{attribute 'GeneratedUsingTerminal: EL2044-0000-0016'}
{attribute addProperty BoxType "EL2044-0000-0016"}
{attribute addProperty Id "Channel_1AT %Q*Channel_D623F56C1Channel_2AT %Q*Channel_D623F56C1Channel_3AT %Q*Channel_D623F56C1Channel_4AT %Q*Channel_D623F56C1"}
{attribute addProperty CRC "4185148518"}
{attribute addProperty Size "4"}
TYPE DIG_Outputs_F9744C66 :
STRUCT
	{attribute addProperty Name "Channel_1"}
	Channel_1 AT %Q* : Channel_D623F56C;
	{attribute addProperty Name "Channel_2"}
	Channel_2 AT %Q* : Channel_D623F56C;
	{attribute addProperty Name "Channel_3"}
	Channel_3 AT %Q* : Channel_D623F56C;
	{attribute addProperty Name "Channel_4"}
	Channel_4 AT %Q* : Channel_D623F56C;
END_STRUCT
END_TYPE

(* stored: Version 1.2.0.0, ProductVersion 3.1.4024.9
   DUT DIG_Outputs_F9744C66: Id {eea1eb29-67e5-4343-9e02-a341537a971c} *)
